(* IEC 61131-3 sources: CodesysTest/export/Function Blocks/SolenoidValves/FB_SingleSolenoidNormallyRetractedActuator.pou/ExtendAsserted.prop, 1 file *)

(* ---- Get.pm.st ---- *)
(*#-#-#-#-#-#-#-#-#-#---Declaration---#-#-#-#-#-#-#-#-#-#-#-#-#*)

VAR
END_VAR
(*#-#-#-#-#-#-#-#-#-#---Implementation---#-#-#-#-#-#-#-#-#-#-#-#-#*)

ExtendAsserted := solenoid0;
